(* CODESYS project CmpTemplate.library
   Title: CmpTemplate
   Version: 3.5.6.0
   Company: OEM

Project tree, tasks and I/O mapping:
  function block MyExternalFunctionblock [ST]: FB_Reinit, FB_Init, FB_Exit, PropTest, MyMethod, MySleep, MyGenerateException
  function MyExternalFunction [ST]
*)

// MyExternalFunctionblock
// Generated comment for MyExternalFunctionblock
FUNCTION_BLOCK MyExternalFunctionblock
VAR_INPUT
	//Partmeter to show message box: 1=Message box will be displayed, 0=else
	bShow : BOOL;
	
	// Parameter to select the Icon of the message box: 1=Show error message box, 0=show information message box
	bError : BOOL;	
	
	// Message text to show in the message box
	MessageText : POINTER TO STRING;
END_VAR
VAR_OUTPUT
	// Result of the operation:
	// + 1: Successful
	// + 0: Failed
	Out : DINT;
END_VAR
VAR
	_internalVar : DINT;
	_property : DWORD;
END_VAR

// FB reinit routine
METHOD FB_Reinit : bool
VAR_INPUT
END_VAR
VAR
END_VAR
END_METHOD

// FB init routine
METHOD FB_Init : bool
VAR_INPUT
	bInitRetains: BOOL;
	bInCopyCode: BOOL;
END_VAR
VAR
END_VAR
END_METHOD

// FB exit routine
METHOD FB_Exit : BOOL
VAR_INPUT
	bInCopyCode: BOOL;
END_VAR
VAR
END_VAR
END_METHOD

{attribute 'monitoring':='call'}
PROPERTY PropTest : DWORD
SET
END_SET
GET
END_GET
END_PROPERTY

METHOD MyMethod : BOOL
VAR_INPUT
	dwIn : DWORD;
END_VAR
END_METHOD

METHOD MySleep : BOOL
VAR_INPUT
	dwSleepMs : DWORD;
END_VAR
END_METHOD

METHOD MyGenerateException : BOOL
VAR_INPUT
	dwException : DWORD;
END_VAR
END_METHOD

END_FUNCTION_BLOCK

// MyExternalFunction
// Generated comment for MyExternalFunction
// RETURN: Returns the runtime system error code (see CmpErrors.library)
FUNCTION MyExternalFunction : DINT
VAR_INPUT
	// Dummy parameter
	p1 : DINT;
END_VAR
VAR
END_VAR

END_FUNCTION
